LIN {X -141.869,Y 0.000,Z -242.561,A 90.000,B 90.000,C 0.000} C_DIS
LIN {X -144.015,Y 0.000,Z -242.561,A 90.000,B 90.000,C 0.000} C_DIS
LIN {X -144.015,Y 0.000,Z -235.012,A 90.000,B 90.000,C 0.000} C_DIS
LIN {X -132.568,Y 0.000,Z -235.012,A 90.000,B 90.000,C 0.000} C_DIS
LIN {X -132.540,Y 0.000,Z -234.994,A 90.000,B 90.000,C 0.000} C_DIS
LIN {X -132.540,Y 0.000,Z -227.464,A 90.000,B 90.000,C 0.000} C_DIS
LIN {X -144.015,Y 0.000,Z -227.464,A 90.000,B 90.000,C 0.000} C_DIS
LIN {X -144.015,Y 0.000,Z -219.915,A 90.000,B 90.000,C 0.000} C_DIS
LIN {X -132.540,Y 0.000,Z -219.915,A 90.000,B 90.000,C 0.000} C_DIS
LIN {X -132.540,Y 0.000,Z -212.366,A 90.000,B 90.000,C 0.000} C_DIS
LIN {X -144.015,Y 0.000,Z -212.366,A 90.000,B 90.000,C 0.000} C_DIS
LIN {X -144.015,Y 0.000,Z -204.817,A 90.000,B 90.000,C 0.000} C_DIS
LIN {X -132.540,Y 0.000,Z -204.817,A 90.000,B 90.000,C 0.000} C_DIS
LIN {X -132.540,Y 0.000,Z -197.269,A 90.000,B 90.000,C 0.000} C_DIS
LIN {X -144.015,Y 0.000,Z -197.269,A 90.000,B 90.000,C 0.000} C_DIS
LIN {X -144.015,Y 0.000,Z -189.720,A 90.000,B 90.000,C 0.000} C_DIS
LIN {X -132.540,Y 0.000,Z -189.720,A 90.000,B 90.000,C 0.000} C_DIS
LIN {X -132.540,Y 0.000,Z -182.171,A 90.000,B 90.000,C 0.000} C_DIS
LIN {X -144.015,Y 0.000,Z -182.171,A 90.000,B 90.000,C 0.000} C_DIS
LIN {X -144.015,Y 0.000,Z -174.622,A 90.000,B 90.000,C 0.000} C_DIS
LIN {X -132.540,Y 0.000,Z -174.622,A 90.000,B 90.000,C 0.000} C_DIS
LIN {X -132.540,Y 0.000,Z -167.073,A 90.000,B 90.000,C 0.000} C_DIS
LIN {X -144.015,Y 0.000,Z -167.073,A 90.000,B 90.000,C 0.000} C_DIS
LIN {X -144.015,Y 0.000,Z -159.525,A 90.000,B 90.000,C 0.000} C_DIS
LIN {X -132.540,Y 0.000,Z -159.525,A 90.000,B 90.000,C 0.000} C_DIS
LIN {X -132.540,Y 0.000,Z -151.976,A 90.000,B 90.000,C 0.000} C_DIS
LIN {X -144.015,Y 0.000,Z -151.976,A 90.000,B 90.000,C 0.000} C_DIS
LIN {X -144.015,Y 0.000,Z -144.427,A 90.000,B 90.000,C 0.000} C_DIS
LIN {X -132.540,Y 0.000,Z -144.427,A 90.000,B 90.000,C 0.000} C_DIS
LIN {X -132.540,Y 0.000,Z -136.878,A 90.000,B 90.000,C 0.000} C_DIS
LIN {X -144.015,Y 0.000,Z -136.878,A 90.000,B 90.000,C 0.000} C_DIS
LIN {X -144.015,Y 0.000,Z -129.329,A 90.000,B 90.000,C 0.000} C_DIS
LIN {X -132.540,Y 0.000,Z -129.329,A 90.000,B 90.000,C 0.000} C_DIS
LIN {X -132.540,Y 0.000,Z -121.781,A 90.000,B 90.000,C 0.000} C_DIS
LIN {X -144.015,Y 0.000,Z -121.781,A 90.000,B 90.000,C 0.000} C_DIS
LIN {X -144.015,Y 0.000,Z -114.232,A 90.000,B 90.000,C 0.000} C_DIS
LIN {X -132.540,Y 0.000,Z -114.232,A 90.000,B 90.000,C 0.000} C_DIS
LIN {X -132.540,Y 0.000,Z -106.683,A 90.000,B 90.000,C 0.000} C_DIS
LIN {X -144.015,Y 0.000,Z -106.683,A 90.000,B 90.000,C 0.000} C_DIS
LIN {X -144.015,Y 0.000,Z -99.134,A 90.000,B 90.000,C 0.000} C_DIS
LIN {X -132.540,Y 0.000,Z -99.134,A 90.000,B 90.000,C 0.000} C_DIS
LIN {X -132.540,Y 0.000,Z -91.586,A 90.000,B 90.000,C 0.000} C_DIS
LIN {X -144.015,Y 0.000,Z -91.586,A 90.000,B 90.000,C 0.000} C_DIS
LIN {X -144.015,Y 0.000,Z -84.037,A 90.000,B 90.000,C 0.000} C_DIS
LIN {X -132.540,Y 0.000,Z -84.037,A 90.000,B 90.000,C 0.000} C_DIS
LIN {X -132.540,Y 0.000,Z -76.488,A 90.000,B 90.000,C 0.000} C_DIS
LIN {X -144.015,Y 0.000,Z -76.488,A 90.000,B 90.000,C 0.000} C_DIS
LIN {X -144.015,Y 0.000,Z -68.939,A 90.000,B 90.000,C 0.000} C_DIS
LIN {X -132.540,Y 0.000,Z -68.939,A 90.000,B 90.000,C 0.000} C_DIS
LIN {X -132.540,Y 0.000,Z -61.390,A 90.000,B 90.000,C 0.000} C_DIS
LIN {X -144.015,Y 0.000,Z -61.390,A 90.000,B 90.000,C 0.000} C_DIS
LIN {X -144.015,Y 0.000,Z -53.842,A 90.000,B 90.000,C 0.000} C_DIS
LIN {X -132.540,Y 0.000,Z -53.842,A 90.000,B 90.000,C 0.000} C_DIS
LIN {X -132.540,Y 0.000,Z -46.293,A 90.000,B 90.000,C 0.000} C_DIS
LIN {X -144.015,Y 0.000,Z -46.293,A 90.000,B 90.000,C 0.000} C_DIS
LIN {X -144.015,Y 0.000,Z -38.744,A 90.000,B 90.000,C 0.000} C_DIS
LIN {X -132.540,Y 0.000,Z -38.744,A 90.000,B 90.000,C 0.000} C_DIS
LIN {X -132.540,Y 0.000,Z -31.195,A 90.000,B 90.000,C 0.000} C_DIS
LIN {X -144.015,Y 0.000,Z -31.195,A 90.000,B 90.000,C 0.000} C_DIS
LIN {X -144.015,Y 0.000,Z -23.646,A 90.000,B 90.000,C 0.000} C_DIS
LIN {X -132.540,Y 0.000,Z -23.646,A 90.000,B 90.000,C 0.000} C_DIS
LIN {X -132.540,Y 0.000,Z -16.098,A 90.000,B 90.000,C 0.000} C_DIS
LIN {X -144.015,Y 0.000,Z -16.098,A 90.000,B 90.000,C 0.000} C_DIS
LIN {X -144.015,Y 0.000,Z -8.549,A 90.000,B 90.000,C 0.000} C_DIS
LIN {X -132.540,Y 0.000,Z -8.549,A 90.000,B 90.000,C 0.000} C_DIS
LIN {X -132.540,Y 0.000,Z -1.000,A 90.000,B 90.000,C 0.000} C_DIS
LIN {X -144.015,Y 0.000,Z -1.000,A 90.000,B 90.000,C 0.000} C_DIS
LIN {X -145.015,Y 0.000,Z 0.000,A 90.000,B 90.000,C 0.000} C_DIS
LIN {X -131.540,Y 0.000,Z 0.000,A 90.000,B 90.000,C 0.000} C_DIS
LIN {X -131.540,Y 0.000,Z -235.536,A 90.000,B 90.000,C 0.000} C_DIS
LIN {X -136.805,Y 0.000,Z -238.969,A 90.000,B 90.000,C 0.000} C_DIS
LIN {X -137.514,Y 0.000,Z -239.368,A 90.000,B 90.000,C 0.000} C_DIS
LIN {X -138.188,Y 0.000,Z -239.825,A 90.000,B 90.000,C 0.000} C_DIS
LIN {X -138.822,Y 0.000,Z -240.335,A 90.000,B 90.000,C 0.000} C_DIS
LIN {X -139.412,Y 0.000,Z -240.895,A 90.000,B 90.000,C 0.000} C_DIS
LIN {X -139.953,Y 0.000,Z -241.502,A 90.000,B 90.000,C 0.000} C_DIS
LIN {X -140.443,Y 0.000,Z -242.152,A 90.000,B 90.000,C 0.000} C_DIS
LIN {X -140.878,Y 0.000,Z -242.840,A 90.000,B 90.000,C 0.000} C_DIS
LIN {X -141.255,Y 0.000,Z -243.561,A 90.000,B 90.000,C 0.000} C_DIS
LIN {X -145.015,Y 0.000,Z -243.561,A 90.000,B 90.000,C 0.000} C_DIS
LIN {X -145.015,Y 0.000,Z 0.000,A 90.000,B 90.000,C 0.000} C_DIS
LIN {X -145.015,Y 5.000,Z 0.000,A 90.000,B 90.000,C 0.000} C_DIS
LIN {X -145.015,Y 75.000,Z 0.000,A 90.000,B 90.000,C 0.000} C_DIS

END
